// TIA Portal V19 export
TYPE "AnalogScale"
   STRUCT
      AnalogMin : Int;
      AnalogMax : Int;
      ScaledMIN : Real;
      ScaledMax : Real;
      ScaledSensor : Real;
   END_STRUCT;
END_TYPE
